// Checks if string is in the format of the IEC-61131 ltime datatype format
FUNCTION F_IsLTime : BOOL
VAR_INPUT
	sValue : REFERENCE TO STRING;
END_VAR
VAR
	i, Length : T_Size;
	pTemp : POINTER TO STRING;
	sLTime_Sharp : STRING := 'LTIME#';
	bHas_D,
	bHas_H,
	bHas_M,
	bHas_S,
	bHas_MS,
	bHas_NS : BOOL;
END_VAR

Length := F_StrLen(ADR(sValue));
pTemp := F_MallocStr(Length+1);
F_StrLCpy(pTemp, ADR(sValue), Length+1);
F_ToUpper(pTemp^);
IF NOT(F_StrNCmp(pTemp^, sLTime_Sharp, 6)) THEN __DELETE(pTemp); RETURN; END_IF
__DELETE(pTemp);

FOR i := 6 TO Length-1 DO
	CASE sValue[i] OF
		68,100: // Check for D/d
			IF NOT F_IsDigit(F_ByteToChar(sValue[i-1])) THEN RETURN; END_IF
			IF bHas_D OR_ELSE bHas_H OR_ELSE bHas_M OR_ELSE bHas_S OR_ELSE bHas_MS OR_ELSE bHas_NS THEN RETURN; END_IF
			bHas_D := TRUE;
		72,104: // Check for H/h
			IF NOT F_IsDigit(F_ByteToChar(sValue[i-1])) THEN RETURN; END_IF
			IF bHas_H OR_ELSE bHas_M OR_ELSE bHas_S OR_ELSE bHas_MS OR_ELSE bHas_NS THEN RETURN; END_IF
			bHas_H := TRUE;
		77,109: // Check for M/m
			IF NOT F_IsDigit(F_ByteToChar(sValue[i-1])) THEN RETURN; END_IF
			IF sValue[i+1] = 83 OR_ELSE sValue[i+1] = 115 THEN
				IF bHas_MS OR_ELSE bHas_NS THEN RETURN; END_IF;
				bHas_MS := TRUE;
			ELSE
				IF bHas_M OR_ELSE bHas_S OR_ELSE bHas_MS OR_ELSE bHas_NS THEN RETURN; END_IF
				bHas_M := TRUE;
				END_IF
		83,115: // Check for S/s
			IF sValue[i-1] = 77 OR_ELSE sValue[i-1] = 109 THEN CONTINUE; END_IF
			IF sValue[i-1] = 78 OR_ELSE sValue[i-1] = 110 THEN CONTINUE; END_IF
			IF NOT F_IsDigit(F_ByteToChar(sValue[i-1])) THEN RETURN; END_IF
			IF bHas_S OR_ELSE bHas_MS OR_ELSE bHas_NS THEN RETURN; END_IF
			bHas_S := TRUE;
		78, 110: // Check for N/n
			IF NOT F_IsDigit(F_ByteToChar(sValue[i-1])) THEN RETURN; END_IF
			IF bHas_NS THEN RETURN; END_IF
			IF sValue[i+1] = 83 OR_ELSE sValue[i+1] = 115 THEN bHas_NS := TRUE; CONTINUE; END_IF
			RETURN;
	ELSE
		IF F_IsDigit(F_ByteToChar(sValue[i])) THEN CONTINUE; END_IF
		RETURN;
	END_CASE
END_FOR
IF F_IsDigit(F_ByteToChar(sValue[i-1])) THEN RETURN; END_IF
F_IsLTime := TRUE;

END_FUNCTION

(* stored: Version 1.1.0.1, ProductVersion 3.1.4024.4
   POU F_IsLTime: Id {d048fade-8caa-4655-83ed-911e9b5c968c}, SpecialFunc None *)
